FUNCTION_BLOCK F_SUB_TOD_TIME (* Subtracts two number values *)
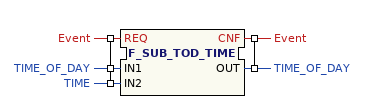
  EVENT_INPUT
    REQ WITH IN1, IN2; (* Normal Execution Request *)
  END_EVENT
  EVENT_OUTPUT
    CNF WITH OUT; (* Execution Confirmation *)
  END_EVENT
  VAR_INPUT
    IN1 : TIME_OF_DAY; (* First funtion input *)
    IN2 : TIME; (* Second function input *)
  END_VAR
  VAR_OUTPUT
    OUT : TIME_OF_DAY; (* Function output *)
  END_VAR
END_FUNCTION_BLOCK
